      |     z = pointintersect[2] + zup
      | 
      |     #apply actual rxryrz to points
      |     # convert the headings to rxryrz and insert those values into the relevant points
      |     rxryrz = convert_heading_to_axang_preheatdown(heading3)
      |     rx = rxryrz[0]
      |     ry = rxryrz[1]
      |     rz = rxryrz[2]
      | 
      |     point1 = p[x + wd1*listleans[0], y + wd1*listleans[1], z + wd1, rx, ry, rz]
      |     point2 = p[x, y, z, rx, ry, rz]
      | 
      |     # convert the headings to rxryrz and insert those values into the relevant points
      |     rxryrz = convert_heading_to_axang(heading3)
      |     rx = rxryrz[0]
      |     ry = rxryrz[1]
      |     rz = rxryrz[2]
      | 
      |     point4 = p[x, y, z, rx, ry, rz]
      |     x = x + l2delxunit * wd2
      |     y = y + l2delyunit * wd2
      |     point5 = p[x, y, z, rx, ry, rz]
      | 
      |     # FIND THE POINTS ON THE LINES OF THE SECOND AROUND PATH
      |     roundoverdistance = 0.05
      |     rod = roundoverdistance * 25.4 / 1000
      | 
      |     # now we have the unit vector. extend the weld distance from the intersection
      |     x = pointintersect[0] + l2delxunit * chamferovermm
      |     y = pointintersect[1] + l2delyunit * chamferovermm
      |     # convert the headings to rxryrz and insert those values into the relevant points
      |     rxryrz = convert_heading_to_axang_ccw(heading3)
      |     rx = rxryrz[0]
      |     ry = rxryrz[1]
      |     rz = rxryrz[2]
      |     point_1 = p[x, y, z, rx, ry, rz]
      | 
      |     x = pointintersect[0] + l2delxunit * rod
      |     y = pointintersect[1] + l2delyunit * rod
      |     point_2 = p[x, y, z, rx, ry, rz]
      | 
      |     # convert the headings to rxryrz and insert those values into the relevant points
      |     rxryrz = convert_heading_to_axang_ccw(heading1)
      |     rx = rxryrz[0]
      |     ry = rxryrz[1]
      |     rz = rxryrz[2]
      | 
      |     x = pointintersect[0] + l1delxunit * rod
      |     y = pointintersect[1] + l1delyunit * rod
      |     point_4 = p[x, y, z, rx, ry, rz]
      | 
      |     # extend the weld distance from the intersection
      |     valid1 = True
      |     # start with the seed
      |     x = pointintersect[0] + l1delxunit * wd3
      |     y = pointintersect[1] + l1delyunit * wd3
      |     point_5 = p[x, y, z, rx, ry, rz]
      |     seed = p[x, y, z, rx, ry, rz]
      |     valid1 = get_inverse_kin_has_solution(seed)
      |     # define the increment
      |     increment = 1.0 # inches
      |     increment = increment * 25.4 / 1000 # meters
      |     while valid1 == True:
      |         wd3 = wd3 + increment
      |         x = pointintersect[0] + l1delxunit * wd3
      |         y = pointintersect[1] + l1delyunit * wd3
      |         seed = p[x, y, z, rx, ry, rz]
      |         valid1 = get_inverse_kin_has_solution(seed)
      |     end
      |     # move back 1 to get the highest valid wd3
      |     # move back 3 to get the third highest valid wd3
      |     wd3 = wd3 - (3.0 * increment)
      |     x = pointintersect[0] + l1delxunit * wd3
      |     y = pointintersect[1] + l1delyunit * wd3
      |     point_5 = p[x, y, z, rx, ry, rz]
      | 
      |     #FIND POINT 3
      |     # by calling analyze_touchpoints()
      |     atret = analyze_touchpoints(point_2, point_1, point_4, point_5, pointintersect)
      |     point_3 = atret[5]
      |     #point 3 will not have the correct rxryrz though because now the gun needs to be face up
      |     rxryrz = convert_heading_to_axang_ccw(heading2)
      |     rx = rxryrz[0]
      |     ry = rxryrz[1]
      |     rz = rxryrz[2]
      |     point_3 = p[point_3[0], point_3[1], point_3[2], rx, ry, rz]
      | 
      |     struct2 = struct(point1=point1, point2=point2, point4=point4, point5=point5, point_1=point_1, point_2=point_2, point_3=point_3, point_4=point_4, point_5=point_5)
      |     return struct2
      | end
      | 
      | # this function analyzes the vertical points
      | # calculates the slope of the edge in question
      | # specifically, for each inch up in the z direction, what is the change in x and change in y direction
      | # returns a list of [nx, ny]
      | def analyze_vertical_touchpoints(p11, p12, p13, p21, p22, p23, p3):
      |     # first, find the equations of the planes from the 6 points
      |     plane1 = findplane(p11, p12, p13)
      |     plane2 = findplane(p21, p22, p23)
      |     # Find the Direction Vector of the Line: The direction vector d of the line of intersection can be found by taking the cross product of the normal vectors of each plane (a, b, and c)
      |     nx = plane1[1]*plane2[2] - plane1[2]*plane2[1]
      |     ny = plane1[2]*plane2[0] - plane1[0]*plane2[2]
      |     nz = plane1[0]*plane2[1] - plane1[1]*plane2[0]
      |     # normalize the vector so the z length is 1
      |     multiplier = 1 / nz
      |     nx = nx * multiplier
      |     ny = ny * multiplier
      |     nz = nz * multiplier # should become equal to 1
      |     ret = [nx, ny]
      |     return ret
      | end
      | 
      | # given 3 points, this finds the plane and its equation
      | # rereturns ax + by + cz + d = 0 in a list of [a, b, c, d]
      | def findplane(p11, p12, p13):
      |     # extract coordinates
      |     x1 = p11[0]
      |     y1 = p11[1]
      |     z1 = p11[2]
      |     x2 = p12[0]
      |     y2 = p12[1]
      |     z2 = p12[2]
      |     x3 = p13[0]
      |     y3 = p13[1]
      |     z3 = p13[2]
      |     # create vectors from the points
      |     v1x = x2-x1
      |     v1y = y2-y1
      |     v1z = z2-z1
      |     v2x = x3-x1
      |     v2y = y3-y1
      |     v2z = z3-z1
      |     #calculate the normal vector using the cross product
      |     nx = v1y*v2z - v1z*v2y # i component
      |     ny = v1z*v2x - v1x*v2z # j component
      |     nz = v1x*v2y - v1y*v2x # k component
      |     # calculate d in the plane equation
      |     d = -1 * (nx*x1 + ny*y1 + nz*z1)
      |     ret = [nx, ny, nz, d]
      |     return ret
      | end
      | 
      | # given a heading, (ccw from +x axis), find the mx+b slope
      | # fails if exactly vertical
      | def get_slope_from_heading(heading):
      |     return tan(heading)
      | end
      | 
      | 
      | 
      | # this function finds the points (and rxryrz) of the 2 points (start and end) of vertical weld section
      | def find_vertical_points(pointintersect, l1delxunit, l1delyunit, l2delxunit, l2delyunit, offset, wd, heading1, heading3):
      | 
      |   # find right side stuff
      |   # find the point in 3d space that is .375 up and .375 over
      |   x = pointintersect[0] + l1delxunit * offset
      |   y = pointintersect[1] + l1delyunit * offset
      |   z = pointintersect[2] + offset
      |   # find rxryrz
      |   rxryrz = convert_heading_to_axang_preheatup(heading1)
      |   rx = rxryrz[0]
      |   ry = rxryrz[1]
      |   rz = rxryrz[2]
      |   path2r1 = p[x, y, z, rx, ry, rz]
      |   path2r2 = p[x, y, z + wd, rx, ry, rz]
      | 
      |   # find left side
      |   # find the point in 3d space that is .375 up and .375 over
      |   x = pointintersect[0] + l2delxunit * offset
      |   y = pointintersect[1] + l2delyunit * offset
      |   z = pointintersect[2] + offset
      |   # find rxryrz
      |   rxryrz = convert_heading_to_axang_preheatup(heading3)
      |   rx = rxryrz[0]
      |   ry = rxryrz[1]
      |   rz = rxryrz[2]
      |   path2l1 = p[x, y, z, rx, ry, rz]
      |   path2l2 = p[x, y, z + wd, rx, ry, rz]
      | 
      |   ret = struct(path2r1=path2r1, path2r2=path2r2, path2l1=path2l1, path2l2=path2l2)
      |   return ret
      | end
      | 
      | # this function converts a unit vector to its heading angle ccw from x+ axis
      | # takes uvx and uvy
      | # returns heading in radians
      | def convert_uv_to_heading(uvx, uvy):
      |   baseang = atan(uvy/uvx)
      |   if uvx < 0:
      |     ang = baseang + pi
      |   elif uvy < 0:
      |     ang = baseang + pi * 2
      |   else:
      |     ang = baseang
      |   end
      |   return ang
      | end
      | 
      | # this function finds the equation of a line, perpendicular to a given line, and going through a given point
      | # takes 3 arguments: m (the original line's slope), x (point's x coord), y (point's y coord). the b of the original line is not needed
      | # returns a list of [m,b] (the slope and intercept of the new line)
      | def find_perpendicular_line(origm, x, y):
      |   m = (1/origm) * -1
      |   b = y - m*x
      |   ret = [m, b]
      |   return ret
      | end
      | 
      | # this function finds the intersection point between two lines in the xy plane
      | # takes 4 arguments: m1, b1, m2, b2
      | # returns a list of [x,y] (the point of intersection)
      | def find_intersection(m1, b1, m2, b2):
      |   # m1x+b1 = m2x+b2
      |   # m1x - m2x = b2 - b1
      |   # x = (b2-b1) / (m1-m2)
      |   x = (b2-b1) / (m1-m2)
      |   y = m1 * x + b1
      |   ret = [x, y]
      |   return ret
      | end
      | 
      | # this function finds the distance between 2 points in 3d space
      | # it takes 6 arguments: x1, y1, z1, x2, y2, z2
      | # it returns a distance
      | def distance_between(x1, y1, z1, x2, y2, z2):
      |   distsquared = (x2-x1)*(x2-x1)+(y2-y1)*(y2-y1)+(z2-z1)*(z2-z1)
      |   dist = sqrt(distsquared)
      |   return dist
      | end
      | 
      | # this function takes a point, a unit vector, and a distance, and adds the distance to the point in the direction of the unit vector (3d space)
      | # it returns a point as a list of coordinates
      | def add_vectordistance_to_point(xi, yi, zi, uvx, uvy, uvz, delta):
      |   xf = xi + uvx * delta
      |   yf = yi + uvy * delta
      |   zf = zi + uvz * delta
      |   ret = [xf, yf, zf]
      |   return ret
      | end
      | 
      | # this function converts a heading (ccw radians from the positive x axis) into rxryrz to be put into a point p[]
      | # this will point the gun in this heading with the bottom side of the gun facing up.
      | # the values used in this program were calculated by doing rotation matrix math in the file on WI-CALVINB10 C. Documents. Theory for converting rotations into axis angle representations
      | def convert_heading_to_axang(heading):
      |  axisxraw = -1 * sin(heading)
      |  axisyraw = cos(heading) + 1
      |  axiszraw = sin(heading)
      | 
      |  magnitude = sqrt(axisxraw*axisxraw + axisyraw*axisyraw + axiszraw*axiszraw)
      | 
      |  axisxunit = axisxraw / magnitude
      |  axisyunit = axisyraw / magnitude
      |  axiszunit = axiszraw / magnitude
      | 
      |  angle = acos( (cos(heading) - 1) / 2 )
      | 
      |  rxout = axisxunit * angle
      |  ryout = axisyunit * angle
      |  rzout = axiszunit * angle
      | 
      |  return [rxout, ryout, rzout]
      | end
      | 
      | # this function converts a heading (ccw radians from the positive x axis) into rxryrz to be put into a point p[]
      | # this will point the gun in this heading with the preheat side of the gun tip facing up. Used for welding in a vertical path.
      | # the values used in this program were calculated by doing rotation matrix math in the file on WI-CALVINB10 C. Documents. Theory for converting rotations into axis angle representations
      | def convert_heading_to_axang_preheatup(heading):
      |  axisxraw = -sin(heading) + 1
      |  axisyraw = cos(heading)
      |  axiszraw = cos(heading)
      | 
      |  magnitude = sqrt(axisxraw*axisxraw + axisyraw*axisyraw + axiszraw*axiszraw)
      | 
      |  axisxunit = axisxraw / magnitude
      |  axisyunit = axisyraw / magnitude
      |  axiszunit = axiszraw / magnitude
      | 
      |  angle = acos( (-sin(heading) - 1) / 2 )
      | 
      |  rxout = axisxunit * angle
      |  ryout = axisyunit * angle
      |  rzout = axiszunit * angle
      | 
      |  return [rxout, ryout, rzout]
      | end
      | 
      | # this function converts a heading (ccw radians from the positive x axis) into rxryrz to be put into a point p[]
      | # this will point the gun in this heading with the preheat side of the gun tip facing down. Used for welding in a vertical path downwards.
      | # the values used in this program were calculated by doing rotation matrix math in the file on WI-CALVINB10 C. Documents. Theory for converting rotations into axis angle representations
      | def convert_heading_to_axang_preheatdown(heading):
      |  axisxraw = -sin(heading) - 1
      |  axisyraw = cos(heading)
      |  axiszraw = -cos(heading)
      | 
      |  magnitude = sqrt(axisxraw*axisxraw + axisyraw*axisyraw + axiszraw*axiszraw)
      | 
      |  axisxunit = axisxraw / magnitude
      |  axisyunit = axisyraw / magnitude
      |  axiszunit = axiszraw / magnitude
      | 
      |  angle = acos( (sin(heading) - 1) / 2 )
      | 
      |  rxout = axisxunit * angle
      |  ryout = axisyunit * angle
      |  rzout = axiszunit * angle
      | 
      |  return [rxout, ryout, rzout]
      | end
      | 
      | # this function converts a heading (ccw radians from the positive x axis) into rxryrz to be put into a point p[]
      | # this will point the gun in this heading with the preheat side of the gun tip facing right. Used for welding counterclockwise around the box.
      | # the values used in this program were calculated by doing rotation matrix math in the file on WI-CALVINB10 C. Documents. Theory for converting rotations into axis angle representations
      | def convert_heading_to_axang_ccw(heading):
      |  axisxraw = -sin(heading)
      |  axisyraw = cos(heading) - 1
      |  axiszraw = -sin(heading)
      | 
      |  magnitude = sqrt(axisxraw*axisxraw + axisyraw*axisyraw + axiszraw*axiszraw)
      | 
      |  axisxunit = axisxraw / magnitude
      |  axisyunit = axisyraw / magnitude
      |  axiszunit = axiszraw / magnitude
      | 
      |  angle = acos( (-cos(heading) - 1) / 2 )
      | 
      |  rxout = axisxunit * angle
      |  ryout = axisyunit * angle
      |  rzout = axiszunit * angle
      | 
      |  return [rxout, ryout, rzout]
      | end
      | 
      | # this function is for getting the points along the path of the corner homing 45
      | # point0 is the point where they touched
      | def get_corner_homing_45_pathpoints(point0):
      |   p0x = point0[0]
      |   p0y = point0[1]
      |   p0z = point0[2]
      |   p0rx = point0[3]
      |   p0ry = point0[4]
      |   p0rz = point0[5]
      | 
      |   #constants
      |   #distances of how far away from point the touchpoints are
      |   d0 = 0.10 # how far from the box to retreat and approach
      |   d1 = 0.03 # first distance from init point
      |   d2 = 0.15 # second distance from init point
      |   d3 = 0.125 #vertical distance from first point
      |   sqrt2 = 0.707106781 # 1/sqrt(2) , the inverse of the sqrt(2)
      | 
      |   ph1 = p[p0x + d0, p0y, p0z + d1, p0rx, p0ry, p0rz] #approach point for turn
      | 
      |   ph2 = p[p0x+d0-d0*0.5-sqrt2*d1, p0y+d0*0.5+sqrt2*d1, p0z+d1, 1.446, -0.8, -0.733]
      |   ph3 = p[p0x+d0-d0*0.5-sqrt2*d2, p0y+d0*0.5+sqrt2*d2, p0z+d1, 1.446, -0.8, -0.733]
      |   ph4 = p[p0x+d0-d0*0.5-sqrt2*d1, p0y-d0*0.5-sqrt2*d1, p0z+d1, 0.626, -1.993, -1.813]
      |   ph5 = p[p0x+d0-d0*0.5-sqrt2*d2, p0y-d0*0.5-sqrt2*d2, p0z+d1, 0.626, -1.993, -1.813]
      | 
      |   # go back to ph1
      |   ph6 = p[p0x + d0, p0y, p0z -0.05, 0, 0, 0] # approach point for under turn
      |   # moveL from ph1 to ph6
      |   ph7 = p[p0x-d1, p0y, p0z-0.05, 0, 0, 0]
      | 
      |   # add the vertical touch points
      |   ph2up = p[ph2[0], ph2[1], ph2[2]+d3, ph2[3], ph2[4], ph2[5]]
      |   ph4up = p[ph4[0], ph4[1], ph4[2]+d3, ph4[3], ph4[4], ph4[5]]
      |   ret = struct(ph1=ph1, ph2=ph2, ph3=ph3, ph4=ph4, ph5=ph5, ph6=ph6, ph7=ph7, ph2up=ph2up, ph4up=ph4up)
      |   is_robot_at_reachable_spot(point0, ret)
      |   return ret
      | end
      | 
      | # this function checks whether the touchpoints are reachable AKA is the robot positioned in the right spot
      | # if everything looks good, it continues.
      | # if it detects a problem, it infinite loops a popup
      | def is_robot_at_reachable_spot(point0, struct_touchpoints):
      |   # first, check whether the corner is too low to the ground that the bottom homing will hit the ground (z < -350)
      |   if point0[2] < -0.350:
      |     # bad
      |     popuptext = "Tank Corner is too low to the ground. Collisions will occur. Stop Program and raise tank. "
      |     # infinite loop
      |     while 1==1:
      |       popup(popuptext, title="Robot Positioning Warning",blocking=True)
      |     end
      |   end
      | 
      | 
      | 
      |   # next, check whether the touchpoints are reachable
      |   structlength = 9
      |   i = 0
      |   allvalid = True
      |   listproblems = ""
      |   listnames = ["ph1", "ph2", "ph3", "ph4", "ph5", "ph6", "ph7", "ph2up", "ph4up"]
      |   while i < structlength:
      |     curr = struct_touchpoints[i]
      |     valid = get_inverse_kin_has_solution(curr)
      |     if not valid:
      |       allvalid = False
      |       listproblems = listproblems + listnames[i]
      |     end
      |     i = i + 1
      |   end
      | 
      |   if not allvalid:
      |     # display
      |     popuptext = "Robot is too far from tank corner. Cannot reach some necessary positions. Stop Program and move robot closer. " + listproblems
      |     # infinite loop
      |     while 1==1:
      |       popup(popuptext, title="Robot Positioning Warning",blocking=True)
      |     end
      |   end
      | 
      | end
      | 
      | # checks the validity of all points during a left weld
      | def check_validity_left(struct1, struct2):
      |   #first, check whether robot is too close
      |   pointintersect = struct1[0]
      |   # next, check if the corner is too close to the robot to do a left around weld (complex but approximately X > -1300)
      |   # if y < 0, then x < -1300. if y < 480, then y > (1300+x)*8. if y > 480, then y > (1235+x)*4 + 500
      |   toocloseleftweld = False
      |   if pointintersect[1] < 0:
      |     if pointintersect[0] > -1.300:
      |       toocloseleftweld = True
      |     end
      |   elif pointintersect[1] < 0.480:
      |     if pointintersect[1] < (1.300 + pointintersect[0])*8:
      |       toocloseleftweld = True
      |     end
      |   else:
      |     if pointintersect[1] < (1.235 + pointintersect[0])*4 + 0.500:
      |       toocloseleftweld = True
      |     end
      |   end
      |   if toocloseleftweld:
      |     # bad
      |     popuptext = "Robot is too close to tank corner. Collisions may occur. Stop Program and move robot farther. "
      |     # infinite loop
      |     while 1==1:
      |       popup(popuptext, title="Robot Positioning Warning",blocking=True)
      |     end
      |   end
      | 
      |   #next, check whether all the points in the weldpath are valid
      |   structlength = 9
      |   i = 0
      |   allvalid = True
      |   listproblems = ""
      |   listnames = ["point1", "point2", "point4", "point5", "point_1", "point_2", "point_3", "point_4", "point_5"]
      |   while i < structlength:
      |     curr = struct2[i]
      |     valid = get_inverse_kin_has_solution(curr)
      |     if not valid:
      |       allvalid = False
      |       listproblems = listproblems + listnames[i]
      |     end
      |     i = i + 1
      |   end
      | 
      |   if not allvalid:
      |     # display
      |     popuptext = "Robot is too far from tank corner. Cannot reach some necessary positions. Stop Program and move robot closer. " + listproblems
      |     # infinite loop
      |     while 1==1:
      |       popup(popuptext, title="Robot Positioning Warning",blocking=True)
      |     end
      |   end
      | 
      | 
      | end
      | 
      | # checks the validity of all points during a right weld
      | def check_validity_right(struct1, struct2):
      |   # first, check whether the right pivot will bonk itself
      |   pointintersect = struct1[0]
      |   heading1 = struct1[1] # this is the direction that the welder will face when doing the right side of the box
      | 
      |   #first, check whether the heading is just too far offset
      |   # more than 15 degrees off of 45 is too much
      |   # normal heading is 216 degrees
      |   #201 degrees to 231 degrees
      |   heading1degrees = heading1 * 180 / pi
      |   if heading1degrees < 201 or heading1degrees > 231 :
      |     # then out of range
      |     popuptext = "Robot is not aligned at a 45 degree angle of corner (15 degree leeway). Collisions may occur. Stop Program and align robot. heading1degrees=" + str_cat("",heading1degrees)
      |     # infinite loop
      |     while 1==1:
      |       popup(popuptext, title="Robot Positioning Warning",blocking=True)
      |     end
      |   end
      | 
      |   #TODO: add the checks for whether x is too close, given the heading
      |   # add checks for whether x is too close, given the heading
      |   # different equations for whether heading offset > 5 degrees or less (inc. negative)
      |   headingoffset = heading1degrees - 216
      |   if headingoffset < 5:
      |     # then calculate a and b
      |     a = 0.4584 + -0.02369 * headingoffset
      |     b = (-1151.4 + 13.83 * headingoffset) / 1000
      |     # check whether x > a*y+b
      |     if pointintersect[0] > a * pointintersect[1] + b:
      |       # bad
      |       popuptext = "Robot is too close to tank corner or not at the right angle. Collisions may occur. Stop Program and align robot. "
      |       # infinite loop
      |       while 1==1:
      |         popup(popuptext, title="Robot Positioning Warning",blocking=True)
      |       end
      |     end
      |   else:
      |     # headingoffset > 5 degrees
      |     if pointintersect[1] < 0:
      |       if pointintersect[0] > -1150.0 / 1000.0:
      |         #bad
      |         popuptext = "Robot is too close to tank corner. Collisions may occur. Stop Program and align robot. "
      |         # infinite loop
      |         while 1==1:
      |           popup(popuptext, title="Robot Positioning Warning",blocking=True)
      |         end
      |       end
      |     else:
      |       # if x > .7736 y - 1101.9 then bad
      |       if pointintersect[0] > 0.7736 * pointintersect[1] - 1101.9 / 1000:
      |         popuptext = "Robot is too close to tank corner. Collisions may occur. Stop Program and align robot. "
      |         # infinite loop
      |         while 1==1:
      |           popup(popuptext, title="Robot Positioning Warning",blocking=True)
      |         end
      |       end
      |     end
      |   end
      | 
      |   #next, check whether all the points in the weldpath are valid
      |   structlength = 9
      |   i = 0
      |   allvalid = True
      |   listproblems = ""
      |   listnames = ["point1", "point2", "point4", "point5", "point_1", "point_2", "point_3", "point_4", "point_5"]
      |   while i < structlength:
      |     curr = struct2[i]
      |     valid = get_inverse_kin_has_solution(curr)
      |     if not valid:
      |       allvalid = False
      |       listproblems = listproblems + listnames[i]
      |     end
      |     i = i + 1
      |   end
      | 
      |   if not allvalid:
      |     # display
      |     popuptext = "Robot is too far from tank corner. Cannot reach some necessary positions. Stop Program and move robot closer. " + listproblems
      |     # infinite loop
      |     while 1==1:
      |       popup(popuptext, title="Robot Positioning Warning",blocking=True)
      |     end
      |   end
      | end
      | 
      | # this function sends a signal to turn extrusion on
      | def turn_extrusion_on():
      |   # flush the channel
      |   resp0 = send_serial_signal(["u", "r", "?"])
      |   # send the signal
      |   resp1 = send_serial_signal(["u", "R", "1"])
      |   # if resp <> "uR1"
      |   if resp1 != [252,82,49]:
      |     # turn off extrusion and heating. inform calvin
      |     resp2 = send_serial_signal(["u", "R", "0"])
      |     resp3 = send_serial_signal(["u", "H", "0"])
      |     popuptext = "Error code encountered while trying to start extrusion. Find Calvin. "
      |     while 1==1:
      |       popup(popuptext, title="Extrusion Error Code",blocking=True)
      |       popup(resp1, blocking=True)
      |     end
      |   end
      | end
      | 
      | # this function sends a signal and receives a response
      | # signal is a list of 3 strings, 1 character each. first is u. second is the next character. third is final character
      | def send_serial_signal(signal):
      |   signal2char = signal[1]
      |   signal3char = signal[2]
      |   listsignal = [252, get_corr_number(signal2char), get_corr_number(signal3char)]
      |   resp1 = WTSerialBridge.send_command("/dev/ttyUSB0",1200, 8, "None", "One", "None", 1000, "None", "None", listsignal, True)
      |   return resp1
      | end
      | 
      | # this function converts a letter into its ascii number
      | def get_corr_number(letter):
      |   if letter == "A":
      |     return 65
      |   elif letter == "H":
      |     return 72
      |   elif letter == "R":
      |     return 82
      |   elif letter == "M":
      |     return 77
      |   elif letter == "E":
      |     return 69
      |   elif letter == "a":
      |     return 97
      |   elif letter == "b":
      |     return 98
      |   elif letter == "h":
      |     return 104
      |   elif letter == "r":
      |     return 114
      |   elif letter == "s":
      |     return 115
      |   elif letter == "m":
      |     return 109
      |   elif letter == "0":
      |     return 48
      |   elif letter == "1":
      |     return 49
      |   elif letter == "2":
      |     return 50
      |   elif letter == "3":
      |     return 51
      |   elif letter == "4":
      |     return 52
      |   elif letter == "5":
      |     return 53
      |   elif letter == "6":
      |     return 54
      |   elif letter == "7":
      |     return 55
      |   elif letter == "8":
      |     return 56
      |   elif letter == "9":
      |     return 57
      |   elif letter == "?":
      |     return 63
      |   end
      | end
      | 
      | # this function checks whether the welder is in the ready state.
      | # to be called at the beginning of Main Program
      | def welder_state_ready():
      |   # flush the channel
      |   resp0 = send_serial_signal(["u", "s", "?"])
      |   # send the signal
      |   resp1 = send_serial_signal(["u", "s", "?"])
      |   # if resp1 == [252,115,49] (us1) then it is ready. otherwise, it is not
      |   if resp1 != [252,115,49]:
      |     popuptext = "Welder is not ready for extrusion. Follow the instructions to start heating welder. "
      |     while 1==1:
      |       popup(popuptext, title="Welder Not Ready",blocking=True)
      |     end
      |   end
      | 
      | end
  path_pre := get_corner_homing_45_pathpoints(tp,tcp_pose_top)
  ph1 := path_pre[0]
  ph2 := path_pre[1]
  ph3 := path_pre[2]
  ph4 := path_pre[3]
  ph5 := path_pre[4]
  ph6 := path_pre[5]
  ph7 := path_pre[6]
  ph2up := path_pre[7]
  ph4up := path_pre[8]
  MoveL speed 250 mm/s, acceleration 200 mm/s^2 (useActiveTCP=true optimoveEnabled=false optiMoveSpeed=0.3 optiMoveAcceleration=0.09) feature=Base
    Waypoint Variable (Variable): variable=ph1
    Waypoint Variable (Variable): variable=ph2
  MoveL speed 20 mm/s, acceleration 100 mm/s^2 (useActiveTCP=true optimoveEnabled=false optiMoveSpeed=0.3 optiMoveAcceleration=0.09) feature=Base
    MoveDirectionNode expression=[-1,-1.0,0.0]
      Until TOOL_CONTACT_DETECTION (allowActions=false retraction=0 decelerationAcceleration=3 decelerationAngularAcceleration=34.906585)
  p11 := get_actual_tcp_pose()
  MoveJ speed 60 deg/s, acceleration 80 deg/s^2 (useActiveTCP=true optimoveEnabled=false optiMoveSpeed=0.3 optiMoveAcceleration=0.09) feature=Base
    Waypoint Variable (Variable): variable=ph2
    Waypoint Variable (Variable): variable=ph2up
  MoveL speed 20 mm/s, acceleration 100 mm/s^2 (useActiveTCP=true optimoveEnabled=false optiMoveSpeed=0.3 optiMoveAcceleration=0.09) feature=Base
    MoveDirectionNode expression=[-1,-1.0,0.0]
      Until TOOL_CONTACT_DETECTION (allowActions=false retraction=0 decelerationAcceleration=3 decelerationAngularAcceleration=34.906585)
  p13 := get_actual_tcp_pose()
  MoveJ speed 60 deg/s, acceleration 80 deg/s^2 (useActiveTCP=true optimoveEnabled=false optiMoveSpeed=0.3 optiMoveAcceleration=0.09) feature=Base
    Waypoint Variable (Variable): variable=ph2up
    Waypoint Waypoint_22: TCP in base x=-454.801 y=459.794 z=358.43 mm, rx=1.4675 ry=-0.379 rz=-0.6081 rad; joints [-90.5, -67.281, 114.422, -41.069, -54.483, -10.697] deg; TCP offset x=-1.032 y=-18.062 z=285.234 mm, rx=0 ry=0 rz=0 rad
    Waypoint Variable (Variable): variable=ph3
  MoveL speed 20 mm/s, acceleration 100 mm/s^2 (useActiveTCP=true optimoveEnabled=false optiMoveSpeed=0.3 optiMoveAcceleration=0.09) feature=Base
    MoveDirectionNode expression=[-1,-1.0,0.0]
      Until TOOL_CONTACT_DETECTION (allowActions=false retraction=0 decelerationAcceleration=3 decelerationAngularAcceleration=34.906585)
  p12 := get_actual_tcp_pose()
  MoveJ speed 60 deg/s, acceleration 80 deg/s^2 (useActiveTCP=true optimoveEnabled=false optiMoveSpeed=0.3 optiMoveAcceleration=0.09) feature=Base
    Waypoint Variable (Variable): variable=ph3
    Waypoint Waypoint_4: TCP in base x=-658.265 y=299.53 z=30.91 mm, rx=0.4268 ry=-1.6215 rz=0.4371 rad; joints [-77.363, -55.591, 142.792, -102.186, -19.322, 105.94] deg; TCP offset x=0 y=0 z=246 mm, rx=0 ry=0 rz=0 rad
  MoveJ speed 60 deg/s, acceleration 80 deg/s^2 (useActiveTCP=true optimoveEnabled=false optiMoveSpeed=0.3 optiMoveAcceleration=0.09) feature=Base
    Waypoint Waypoint_5: TCP in base x=-448.863 y=524.6 z=-175.967 mm, rx=2.4733 ry=-1.8744 rz=0.2053 rad; joints [-65.056, -57.525, 139.86, -164.756, -91.924, 99.291] deg
    SuppressedNode
      Waypoint Waypoint_5: TCP in base x=-542.919 y=212.782 z=86.75 mm, rx=-0.746 ry=-1.5701 rz=-0.8083 rad; joints [-15.32, -63.738, 160.053, -88.648, -229.235, 89.501] deg
    Waypoint Waypoint_10: TCP in base x=-559.13 y=259.234 z=102.446 mm, rx=-0.8226 ry=-1.4861 rz=-0.8815 rad; joints [-31.871, -61.56, 166.811, -101.777, -239.831, 87.599] deg; TCP offset x=-1.157 y=-95.604 z=257.595 mm, rx=0 ry=0 rz=0 rad
  MoveJ speed 60 deg/s, acceleration 80 deg/s^2 (useActiveTCP=true optimoveEnabled=false optiMoveSpeed=0.3 optiMoveAcceleration=0.09) feature=Base
    Waypoint Variable (Variable): variable=ph4
  MoveL speed 20 mm/s, acceleration 100 mm/s^2 (useActiveTCP=true optimoveEnabled=false optiMoveSpeed=0.3 optiMoveAcceleration=0.09) feature=Base
    MoveDirectionNode expression=[-1.0,1.0,0.0]
      Until TOOL_CONTACT_DETECTION (allowActions=false retraction=0 decelerationAcceleration=3 decelerationAngularAcceleration=34.906585)
  p21 := get_actual_tcp_pose()
  MoveL speed 250 mm/s, acceleration 1200 mm/s^2 (useActiveTCP=true optimoveEnabled=false optiMoveSpeed=0.3 optiMoveAcceleration=0.09) feature=Base
    Waypoint Variable (Variable): variable=ph4
    Waypoint Variable (Variable): variable=ph4up
  MoveL speed 20 mm/s, acceleration 100 mm/s^2 (useActiveTCP=true optimoveEnabled=false optiMoveSpeed=0.3 optiMoveAcceleration=0.09) feature=Base
    MoveDirectionNode expression=[-1.0,1.0,0.0]
      Until TOOL_CONTACT_DETECTION (allowActions=false retraction=0 decelerationAcceleration=3 decelerationAngularAcceleration=34.906585)
  p23 := get_actual_tcp_pose()
  MoveL speed 250 mm/s, acceleration 1200 mm/s^2 (useActiveTCP=true optimoveEnabled=false optiMoveSpeed=0.3 optiMoveAcceleration=0.09) feature=Base
    Waypoint Variable (Variable): variable=ph4up
    Waypoint Variable (Variable): variable=ph5
  MoveL speed 20 mm/s, acceleration 100 mm/s^2 (useActiveTCP=true optimoveEnabled=false optiMoveSpeed=0.3 optiMoveAcceleration=0.09) feature=Base
    MoveDirectionNode expression=[-1.0,1.0,0.0]
      Until TOOL_CONTACT_DETECTION (allowActions=false retraction=0 decelerationAcceleration=3 decelerationAngularAcceleration=34.906585)
  p22 := get_actual_tcp_pose()
  MoveJ speed 60 deg/s, acceleration 80 deg/s^2 (useActiveTCP=true optimoveEnabled=false optiMoveSpeed=0.3 optiMoveAcceleration=0.09) feature=Base
    Waypoint Variable (Variable): variable=ph5
    Waypoint Variable (Variable): variable=ph4
    SuppressedNode
      Waypoint Waypoint_5: TCP in base x=-542.919 y=212.782 z=86.75 mm, rx=-0.746 ry=-1.5701 rz=-0.8083 rad; joints [-15.32, -63.738, 160.053, -88.648, -229.235, 89.501] deg; TCP offset x=0 y=0 z=246 mm, rx=0 ry=0 rz=0 rad
    Waypoint Waypoint_11: TCP in base x=-559.13 y=259.234 z=102.446 mm, rx=-0.8226 ry=-1.4861 rz=-0.8815 rad; joints [-31.871, -61.56, 166.811, -101.777, -239.831, 87.599] deg; TCP offset x=-1.157 y=-95.604 z=257.595 mm, rx=0 ry=0 rz=0 rad
    Waypoint Waypoint_12: TCP in base x=-448.863 y=524.6 z=-175.967 mm, rx=2.4733 ry=-1.8744 rz=0.2053 rad; joints [-65.056, -57.525, 139.86, -164.756, -91.924, 99.291] deg; TCP offset x=0 y=0 z=246 mm, rx=0 ry=0 rz=0 rad
    Waypoint Waypoint_4: TCP in base x=-658.265 y=299.53 z=30.91 mm, rx=0.4268 ry=-1.6215 rz=0.4371 rad; joints [-77.363, -55.591, 142.792, -102.186, -19.322, 105.94] deg
    Waypoint Waypoint_13: TCP in base x=-343.952 y=632.142 z=615.175 mm, rx=-0.0259 ry=-0.0088 rz=-0.5675 rad; joints [-77.363, -55.591, 142.791, -175.721, 90.298, 134.942] deg
    Waypoint Variable (Variable): variable=ph6
    Waypoint Variable (Variable): variable=ph7
  MoveL speed 20 mm/s, acceleration 100 mm/s^2 (useActiveTCP=true optimoveEnabled=false optiMoveSpeed=0.3 optiMoveAcceleration=0.09) feature=Base
    MoveDirectionNode (selectedDirection=ZPlus)
      Until TOOL_CONTACT_DETECTION (allowActions=false retraction=0 decelerationAcceleration=3 decelerationAngularAcceleration=34.906585)
  p3 := get_actual_tcp_pose()
  MoveJ speed 60 deg/s, acceleration 80 deg/s^2 (useActiveTCP=true optimoveEnabled=false optiMoveSpeed=0.3 optiMoveAcceleration=0.09) feature=Base
    Waypoint Variable (Variable): variable=ph7
    Waypoint Variable (Variable): variable=ph6
    Waypoint Waypoint_14: TCP in base x=-343.952 y=632.142 z=615.175 mm, rx=-0.0259 ry=-0.0088 rz=-0.5675 rad; joints [-77.363, -55.591, 142.791, -175.721, 90.298, 134.942] deg
    Waypoint Waypoint_4: TCP in base x=-658.265 y=299.53 z=30.91 mm, rx=0.4268 ry=-1.6215 rz=0.4371 rad; joints [-77.363, -55.591, 142.792, -102.186, -19.322, 105.94] deg
    Waypoint Waypoint_41: TCP in base x=392.128 y=533.269 z=644.149 mm, rx=0.0578 ry=2.126 rz=2.134 rad; joints [-198.126, -117.852, 133.303, -13.01, -11.421, -6.036] deg; TCP offset x=0 y=-4 z=284 mm, rx=0 ry=0 rz=0 rad
    'above waypoint is home'
  SuppressedNode
    SafeHome (positionOptionType=SPEED_AND_ACCELERATION speed=1.047198 acceleration=1.396263 nextMotionTime=2)
  ''
  ''
  ''
  ''
  ''
  ''
Thread Thread_1 (runOnlyOnce=true)
  Loop While (checkContinuously=false) expression=True
    If freedrive_m_var≟ True
      Script: freedrive_mode()
      free_dr_already := True
    Else 
      If free_dr_already
        Script: end_freedrive_mode()
    Script: sync()
SuppressedNode
  Thread Thread_2 (runOnlyOnce=false)
    Loop While (checkContinuously=false) expression=True
      If thread2trigger≟ True
        'do the dot extrude'
        Wait Sleep waitTime=5
        URCap WireTank Serial (WireTank Serial, WireTank, LLC) dataModel(byte_array=true, NODE_TITLE=Serial Bridge uR1, Command=[252,82,49], QUERY=false, OUTPUT_ENTRY=Static, Variable(key=OUTPUT_VARIABLE, variable(name=HwResp)))
        Wait Sleep waitTime=2
        URCap WireTank Serial (WireTank Serial, WireTank, LLC) dataModel(QUERY=false, NODE_TITLE=Serial Bridge uR0, Command=[252,82,48], byte_array=true, OUTPUT_ENTRY=Static, Variable(key=OUTPUT_VARIABLE, variable(name=HwResp)))
        thread2trigger := False
      Script: sync()
